PROGRAM MAIN
VAR
	Data					: ST_DATA;
	
	
	// ============== Set input/output mode: 	StaticData, SimulinkPlant, VirtualPlant PhysicalPlant	
	EmulatedState 			: E_EmulatedState 		:= E_EmulatedState.VirtualPlant;		
	
END_VAR



//============ UPDATE DAQ =============	
P_UpdateDAQ(Data := Data);

//============ UPDATE HMI =============	
P_UpdateHmi(Data := Data);

END_PROGRAM

(* stored: Version 1.1.0.1, ProductVersion 3.1.4022.11
   POU MAIN: Id {24755970-32eb-41b5-9fc7-46989e4620de}, SpecialFunc None *)
